// TIA Portal V17 export
// export: Created 2022-07-04T13:04:17.8419801Z, ExportSetting WithDefaults, DisplayName Totally Integrated Automation Portal, DisplayVersion V17, DisplayName TIA Portal Openness, DisplayVersion V17, DisplayName TIA Portal Version Control Interface, DisplayVersion V17, DisplayName STEP 7 Professional, DisplayVersion V17, DisplayName STEP 7 Safety, DisplayVersion V17, DisplayName WinCC Advanced, DisplayVersion V17
TYPE "typeOPCUAStatus"
// stored: IsFailsafeCompliant false
   STRUCT
      done : Bool;
      busy : Bool;
      error : Bool;
      status : DWord;
   END_STRUCT;
END_TYPE
